// TIA Portal V18 export
FUNCTION_BLOCK "transfer"   // FB1, FBD
{ S7_Optimized_Access := 'TRUE' }
VERSION : 0.1
// stored: AutoNumber true, IsIECCheckEnabled false, IsRetainMemResEnabled false, MemoryReserve 100, SetENOAutomatically false, UDAEnableTagReadback false
   VAR
      ton_no_con { S7_SetPoint := 'True'} : TON_TIME;
   END_VAR
BEGIN

REGION Network 1: bool
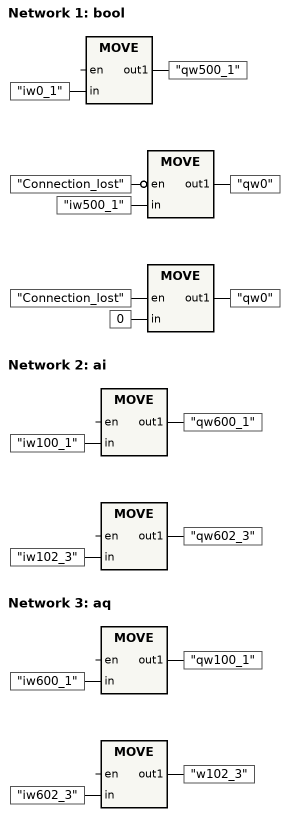
   "qw500_1" := "iw0_1";
   IF NOT "Connection_lost" THEN "qw0" := "iw500_1"; END_IF;
   IF "Connection_lost" THEN "qw0" := 0; END_IF;
END_REGION

REGION Network 2: ai
   "qw600_1" := "iw100_1";
   "qw602_3" := "iw102_3";
END_REGION

REGION Network 3: aq
   "qw100_1" := "iw600_1";
   "w102_3" := "iw602_3";
END_REGION

REGION Network 4: enc
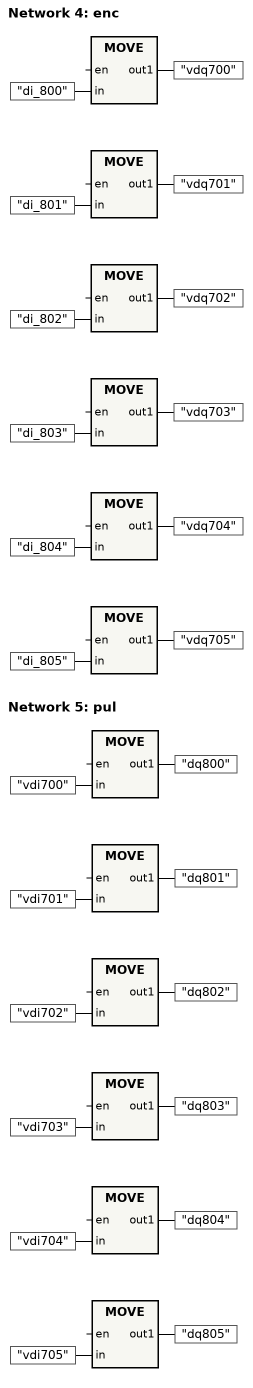
   "vdq700" := "di_800";
   "vdq701" := "di_801";
   "vdq702" := "di_802";
   "vdq703" := "di_803";
   "vdq704" := "di_804";
   "vdq705" := "di_805";
END_REGION

REGION Network 5: pul
   "dq800" := "vdi700";
   "dq801" := "vdi701";
   "dq802" := "vdi702";
   "dq803" := "vdi703";
   "dq804" := "vdi704";
   "dq805" := "vdi705";
END_REGION

REGION Network 6: comms
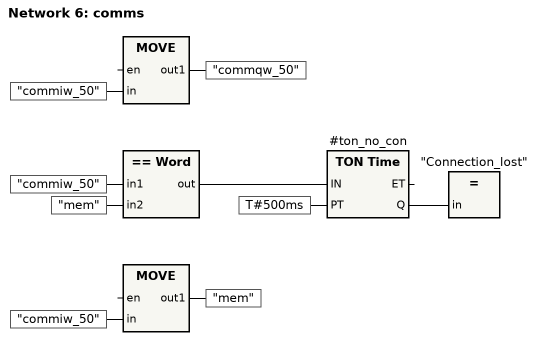
   "commqw_50" := "commiw_50";
   #ton_no_con(IN := "commiw_50" = "mem", PT := T#500ms);   // TON
   "Connection_lost" := #ton_no_con.Q;
   "mem" := "commiw_50";
END_REGION
END_FUNCTION_BLOCK
